RoboDK station: pr52021.rdk

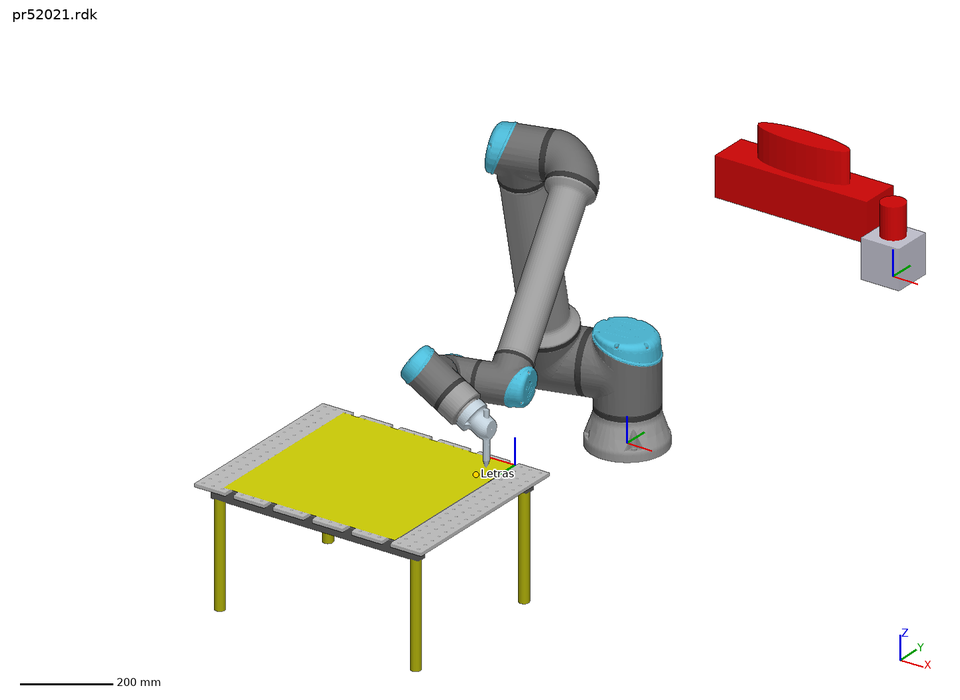
[picture v0: the station drawn from its stored meshes, robots at their saved joint values, targets as dots, program paths as lines]
Station pr52021 (saved by RoboDK 5.2.4). Poses are relative to the parent item; angles as X-Y-Z fixed-axis rotations.
Station parameters (name, value as stored): FRAMELETRAS, RoboDK item (1733015690624) of type 3, TARLETRAS, Pose(41.936, 86.310, -1.006,  0.000, 0.000, -0.000): [[ 1.000, 0.000, 0.000, 41.936 ],  [ -0.000, 1.000, -0.000, 86.310 ],  [ -0.000, 0.000, 1.000, -1.006 ],  [ 0.000, 0.000, 0.000, 1.000 ]] , orden1, 3, Pencil, 0, Palletizing Plugin
  - frame UR10e Base at (0, 0, 0) mm
    - robot UR10e: 6 axes, payload 10 kg, reach 1300 mm, repeatability 0.05 mm, weight 28.9 kg
        modified DH rows (alpha deg, a mm, theta deg, d mm): 0, 0, 0, 180.7; 90, 0, 180, 0; 0, 612.6, 0, 0; 0, 571.335, 0, 174.15; -90, 0, 0, 119.85; 90, 0, 180, 116.55
        joint limits [-360, -360, -360, -360, -360, -360] to [360, 360, 360, 360, 360, 360]; home [0, -90, -90, 0, 90, 0]; saved at [-74.729, -108.388, -106.051, -31.039, 146.663, 118.637]
      - tool Pencil, TCP at (1.16, -82.2, 101.78) mm, rotated rx 0 ry -60 rz 90 deg, size 74.9 x 125 x 107.3 mm
  - object Table at (0, -960, 300) mm, size 596.9 x 482.6 x 304.8 mm, geometry from welding_table.sld
  - object Plane at (0, -970, 307.87) mm, size 450 x 450 x 0.2 mm, geometry from plane_1m.sld
  - program replaceobjects (1 instructions, listed below)
  - Python program SETPARAMS (listed below)
  - frame FrameLetras at (225.65, -744.57, 308.41) mm, rotated rx 0 ry 0 rz 180 deg
    - target Letras (Cartesian target) at (41.94, 86.31, -0.1) mm; joints [-57.054, -144.497, -94.688, 12.474, -43.385, -322.349] of UR10e
  - Python program GETPARAMS (listed below)
  - program Main (3 instructions, listed below)
  - Python program WeldOn (listed below)
  - Python program elipsee (listed below)
  - Python program Parame (listed below)
  - Python program varios (listed below)
  - frame Frame 3 at (0, 1000, 0) mm
    - object box at (0, 0, 0) mm, size 100 x 100 x 100 mm, geometry from box.sld
    - object cil at (0, 0, 100) mm, size 60 x 60 x 80 mm, geometry from part.sld
    - object martillo1_copy at (-340, 150, 100) mm, size 400 x 100 x 180 mm

--- program replaceobjects (robot UR10e) ---
  Replace objects

--- Python program SETPARAMS ---
from robolink import *    # RoboDK API
from robodk import*        # Robot toolbox

RDK = Robolink()

robot = RDK.ItemUserPick('',ITEM_TYPE_ROBOT) 	#adquirir todos los parámetros del robot
if not robot.Valid():
    quit()
reference = robot.Parent()  # devuelve el artículo
robot.setPoseFrame(reference)#establece el marco de referencia de un robot
pose_ref=robot.Pose()  #devuelve la posición actual del robot con matriz
b=robodk.pose_2_xyzrpw(pose_ref) # devuelve la posición actual del robot

frameletras = RDK.Item("FrameLetras",ITEM_TYPE_FRAME)
robot.setPoseFrame(frameletras)

tarletras = RDK.Item("Letras",ITEM_TYPE_TARGET)
tarletras = tarletras.Pose()

ORDEN = 0

RDK.RunProgram("WeldOn(-1)")
RDK.setParam("orden1",ORDEN)
while (ORDEN1 < 3):
    robot.MoveJ(tarletras*roty(-pi))
    robot.MoveJ(tarletras*transl(0,50,0)*roty(-pi))
    robot.MoveJ(tarletras*transl(100,0,50)*roty(-pi))
    ORDEN1+= 1
    RDK.setParam("orden1",ORDEN)

--- Python program GETPARAMS ---
from robolink import *    # RoboDK API
from robodk import*        # Robot toolbox
from time import*
RDK = Robolink()

robot = RDK.ItemUserPick('',ITEM_TYPE_ROBOT) 	#adquirir todos los parámetros del robot
if not robot.Valid():
    quit()
reference = robot.Parent()  # devuelve el artículo
robot.setPoseFrame(reference)#establece el marco de referencia de un robot
pose_ref=robot.Pose()  #devuelve la posición actual del robot con matriz
b=robodk.pose_2_xyzrpw(pose_ref) # devuelve la posición actual del robot

frameletras = RDK.Item("FrameLetras",ITEM_TYPE_FRAME)
robot.setPoseFrame(frameletras)

tarletras = RDK.Item("Letras")
tarletras = tarletras.Pose()


#obtener parametros de otro python desde la estacion
esperaorden = RDK.getParam("orden1")
while (esperaorden < 2):
    esperaorden = RDK.getParam("orden1")
    pass

robot.setSpeed(50,50)
RDK.setSimulationSpeed(0.25)
robot.MoveJ(tarletras*roty(-pi))
RDK.RunProgram("WeldOn(1)")
sleep(0.5)
robot.MoveJ(tarletras*transl(100,50,0)*roty(-pi))
robot.MoveJ(tarletras*transl(0,50,50)*roty(-pi))
RDK.RunProgram("WeldOn(0)")

--- program Main (robot UR10e) ---
  Run SETPARAMS
  Wait orden1=3
  Run GETPARAMS

--- Python program WeldOn ---
# This macro allows simulating the material deposition of a weld gun
# By default, this macro will activate the trace once it is called.
# Run the macro ArcEnd to stop the trace.
#
# The macros ArcStart, ArcEnd and WeldOn, SpindleOn, all behave in a similar way, the only difference is the default behavior
# This behavior simmulates Fanuc Arc Welding and triggers appropriate output when using the customized post processor.
# Select ESC to clear the trace manually.
#
# It is possible to call WeldOn(ON) to simulate turning the material deposition ON or WeldOn(OFF) to stop simulating the gun
# Calling WeldOn(RESET) clears all displayed data.
# The macro will output spray gun statistics
#
# Optional:
#     This macro can manage multiple guns and multiple colors.
#     As an example, you can call this macro the following way:
#
# WeldOn(State, ToolName, Color)
#     State: [ON/OFF/RESET]
#     TorchName: The name of the tool. For example: Tool 1
#     Color: A named color or a hex color in the format: '#AARRGGBB'
#             Important: for full color definition you should provide Alpha channel first
#
# Examples:
#     WeldOn(ON)                 # Turn on the trace using the default color
#     WeldOn(OFF)                # Turn off the tool trace
#     WeldOn(ON, Tool 1, yellow) # Turn on the trace for tool 1 in yellow
#     WeldOn(ON, Tool 2, blue) # Turn on the trace for tool 2 in blue
#     WeldOn(OFF, Torch1)        # Turn off trace for Torch 1
#     WeldOn(ON, Torch1, #889900FF) # Turn on the trace for torch 2 in a violet color
#     WeldOn(ON, ,red)         # Turn on the trace for a generic torch in red color
#
# --------------------------------------------------------------
# This script shows how to create "spray" object in RoboDK that allows simulating particle deposition by using:
# RDK.Spray_Add(tool, object, options_command, volume, geometry)
#    tool: tool item (TCP) to use
#    object: object to project the particles
#    options_command (optional): string to specify options.
#    volume (optional): Matrix of parameters defining the volume of the spray gun
#    geometry (optional): Matrix of vertices defining the triangles.
#
# More information here:
# https://robodk.com/doc/en/PythonAPI/robolink.html#robolink.Robolink.Spray_Add
# https://robodk.com/doc/en/RoboDK-API.html
#
# The scripts ArcStart, ArcEnd and WeldOn and SpindleOn behave in a similar way, the only difference is the default behavior
# This behavior simmulates Fanuc Arc Welding and triggers appropriate output when using the customized post processor.
# Select ESC to clear the trace manually.
#
# Example scripts that use Spray_Add:
#     SpindleOn / SpindleOff    -> Turn trace On/Off
#     ArcOn / ArcOff            -> Turn trace On/Off
#     SprayOn / SprayOff        -> Simulate a spray given a workspace volume (for painting)
#     WeldOn / WeldOff          -> Support for multiple weld guns
#
#----------------------------------------------------------

# Constant variables for the first parameter:
ACTION_RESET    = -1    # Same as: RESET (clear all traces)
ACTION_OFF      =  0    # Same as: OFF (turn on)
ACTION_ON       =  1    # Same as: ON (turn off)

# Define the default Action (ACTION_OFF to deactivate, ACTION_ON to activate, ACTION_RESET to clear any spray gun/trace)
# Setting it to None will display a message
Action = ACTION_ON

# Define the default color as a named color or as #AARRGGBB (Alpha, Red, Green Blue)
# COLOR = 'blue'
COLOR = '#CC3344FF' # AARRGGBB

# Use a specific tool as a spray gun
Tool_Name = "Pencil"    # Use the active tool
#Tool_Name = 'Torch1'

# Use a specific object to project particles:
Object_Name = "Plane"  # Use the first object in the active reference frame
#Object_Name = 'Part'

# --------------------------------------------------
# Program start:
from robolink import *    # API to communicate with RoboDK
from robodk import *      # basic matrix operations
RDK = Robolink()

# quit if we are not in simulation mode
if RDK.RunMode() != RUNMODE_SIMULATE:
    quit()

# Check command input (parameters passed in the call). This is the same as if we were doing a command line call passing parameters.
import sys
if len(sys.argv) > 1:
    Action_str = sys.argv[1].strip().upper()
    if 'ON' in Action_str:
        Action = ACTION_ON
    elif 'OFF' in Action_str:
        Action = ACTION_OFF
    elif 'RESET' in Action_str:
        Action = ACTION_RESET
    else:
        Action = int(Action_str)

    if len(sys.argv) > 2:
        Tool_Name = sys.argv[2].strip()
        if Tool_Name == '':
            Tool_Name = None

        if len(sys.argv) > 3:
            COLOR = sys.argv[3].lower().strip()

# Display summary
print("Applying action: " + str(Action))
print("Using tool: " + str(Tool_Name))
print("Using color: " + COLOR)

# Get any previously added spray gun simulations and display statistics (spray on the part vs spray falling out of the part)
info, data = RDK.Spray_GetStats()
n_sprays = data.size(1)
spray_id = -1
if n_sprays > 0 and Tool_Name is not None:
    spray_id = RDK.getParam(Tool_Name)
    if spray_id is None or Action == ACTION_ON or type(spray_id) == str or spray_id >= n_sprays:
        spray_id = -1

    print("Spray gun statistics:")
    print(info)
    print(data.tr())
    # # Diplay statistics
    # RDK.ShowMessage("Material used: %.1f%%<br>Material waisted: %.1f%%<br>Total particles: %.1f" % (data[1,0],data[2,0],data[3,0]), True)
    # # Clear previous spray
    # RDK.Spray_Clear()


# If the default Action is None, display a message to activate/deactivate the spray gun
if Action is None:
    print('Note: This macro can be called as ArcStart(1) or ArcStart(0) or ArcStart(-1)')
    entry = mbox('Turn gun ON or OFF', ('On', '1'), ('Off', '0'))
    if not entry:
        quit()
    Action = int(entry)

# Apply the desired action
if Action == ACTION_OFF:
    # Turn the gun off
    RDK.Spray_SetState(SPRAY_OFF, spray_id)

elif Action == ACTION_RESET:
    # Clear all spray simulations (same as pressing ESC key)
    RDK.Spray_Clear(spray_id)

elif Action == ACTION_ON:
    # Create a new spray gun object in RoboDK
    # by using RDK.Spray_Add(tool, object, options_command, volume, geometry)
    # tool: tool item (TCP) to use
    # object: object to project the particles
    # options_command (optional): string to specify options. Example:
    #     STEP=AxB: Defines the grid to be projected 1x1 means only one line of particle projection (for example, for welding)
    #     PARTICLE: Defines the shape and size of particle (sphere or particle), unless a specific geometry is provided:
    #       a- SPHERE(radius, facets)
    #       b- SPHERE(radius, facets, scalex, scaley, scalez)
    #       b- CUBE(sizex, sizey, sizez)
    #     RAND=factor: Defines a random factor factor 0 means that the particles are not deposited randomly
    #     ELLYPSE: defines the volume as an ellypse (default)
    #     RECTANGLE: defines the volume as a rectangle
    #     PROJECT: project the particles to the surface (default) (for welding, painting or scanning)
    #     NO_PROJECT: does not project the particles to the surface (for example, for 3D printing)
    #
    # volume (optional): Matrix of parameters defining the volume of the spray gun
    # geometry (optional): Matrix of vertices defining the triangles.

    if spray_id < 0:
        tool = 0    # auto detect active tool
        obj = 0     # auto detect object in active reference frame
        if Tool_Name is not None:
            tool = RDK.Item(Tool_Name, ITEM_TYPE_TOOL)

        if Object_Name is not None:
            obj = RDK.Item(Object_Name, ITEM_TYPE_OBJECT)
        # We can specify a given tool object and/or object
        #robot = RDK.Item("ABB IRB 2600-12/1.85", ITEM_TYPE_ROBOT)
        #tools = robot.Childs()
        #if len(tools) > 0:
        #    tool = tools[0]
        #obj = RDK.Item('object', ITEM_TYPE_OBJECT)

        # Create volume parameters
        options_command = "NO_PROJECT PARTICLE=SPHERE(2,8,1,1,1) STEP=1x0 RAND=0 COLOR=" + COLOR

        spray_id = RDK.Spray_Add(tool, obj, options_command)

    # Remember the ID of the spray gun for later
    if Tool_Name is not None:
        RDK.setParam(Tool_Name, spray_id)

    # Apply the state to activate the trace
    RDK.Spray_SetState(SPRAY_ON, spray_id)

--- Python program elipsee ---
from robolink import *    # RoboDK API
from robodk import *      # Robot toolbox
from time import sleep
RDK = Robolink()
rob = robodk

robot = RDK.ItemUserPick('',ITEM_TYPE_ROBOT)    #adquirir todos los parámetros d el robot
if not robot.Valid():
    quit()
reference = robot.Parent()  # devuelve el artículo robot.setPoseFrame(reference)#establece el marco de referencia de un robot pose_ref=robot.Pose()  #devuelve la posición actual del robot con matriz
robot.setPoseFrame(reference)#establece el marco de referencia de un robot

frameletras = RDK.Item("FrameLetras",ITEM_TYPE_FRAME)
robot.setPoseFrame(frameletras)

def elipse():
    Ref1 = RDK.Item("Letras",ITEM_TYPE_TARGET)
    RefTar = Ref1.Pose()
    b1 = rob.pose_2_xyzrpw(RefTar)
    t = -pi/2
    x0= b1[0]
    y0= b1[1]
    z0= b1[2]
    a=30
    b=10
    RDK.RunProgram('WeldOn(-1)')
    robot.MoveJ(RefTar*roty(-pi))
    robot.setSpeed(2050,2000)
    while (t <=3*pi/2):
        pos = transl(x0 + a*cos(t), y0 + b*sin(t), z0)*roty(-pi)
        robot.MoveJ(pos)
        if (t==-pi/2):
            sleep(2)
            RDK.RunProgram('WeldOn')
        t +=pi/360

elipse()
RDK.RunProgram('WeldOn(0)')

--- Python program Parame ---
from robolink import *    # RoboDK API
from robodk import *      # Robot toolbox
from time import sleep
RDK = Robolink()
rob = robodk

robot = RDK.ItemUserPick('',ITEM_TYPE_ROBOT)    #adquirir todos los parámetros d el robot
if not robot.Valid():
    quit()
reference = robot.Parent()  # devuelve el artículo robot.setPoseFrame(reference)#establece el marco de referencia de un robot pose_ref=robot.Pose()  #devuelve la posición actual del robot con matriz
robot.setPoseFrame(reference)#establece el marco de referencia de un robot

def elipse():
    frameletras = RDK.Item("FrameLetras",ITEM_TYPE_FRAME)
    robot.setPoseFrame(frameletras)
    Ref1 = RDK.Item("Letras",ITEM_TYPE_TARGET)
    RefTar = Ref1.Pose()
    t = -pi/2
    a=20
    b=10
    k = 4
    RDK.RunProgram('WeldOn(-1)')
    robot.MoveJ(RefTar*roty(pi))
    robot.setSpeed(2050,2000)
    while (t <=3*pi/2):
        pos = RefTar*transl(a*cos(t)*k,b*sin(t)*k, 0)*roty(pi)
        robot.MoveJ(pos)
        if (t==-pi/2):
            sleep(2)
            RDK.RunProgram('WeldOn')
        t +=pi/360

elipse()
RDK.RunProgram('WeldOn(0)')

--- Python program varios ---
from robolink import *    # RoboDK API
from robodk import *      # Robot toolbox
from time import*
RDK = Robolink()


# Program example:
item1 = RDK.Item('box')
item2 = RDK.Item('cil')
frame3 = RDK.Item('Frame 3')


if item1.Valid():
    print('Item selected: ' + item1.Name())
    print('Item posistion: ' + repr(item1.Pose()))
    print('Item selected: ' + item2.Name())
    print('Item posistion: ' + repr(item2.Pose()))


print('Items in the station:')
itemlist = RDK.ItemList()
for i in itemlist:
 print(i.Name())

item1.Copy()
item1_Copy = frame3.Paste()

item2.Copy()
item2_Copy = frame3.Paste()
sleep(2)
martillo = RDK.MergeItems(list_items = [item1_Copy,item2_Copy])
martillo.setVisible(False)
posmartillo = martillo.Pose()
martillo.setPose(posmartillo*transl(0,100,0))
martillo.setName("martillo1_copy")
martillo.setVisible(True)
sleep(2)
martillo.Recolor([1,0,0,1])
RDK.ShowMessage("solicitando a usuario... ",False)
pedido = mbox("ingrese valor de escala en x,y,z desde 1 en adelante",entry="1,1,1")
x,y,z = [int(x.replace(' ','')) for x in  pedido.split(',')]
martillo.Scale([x,y,z])
RDK.ShowMessage("fin de programa ")
